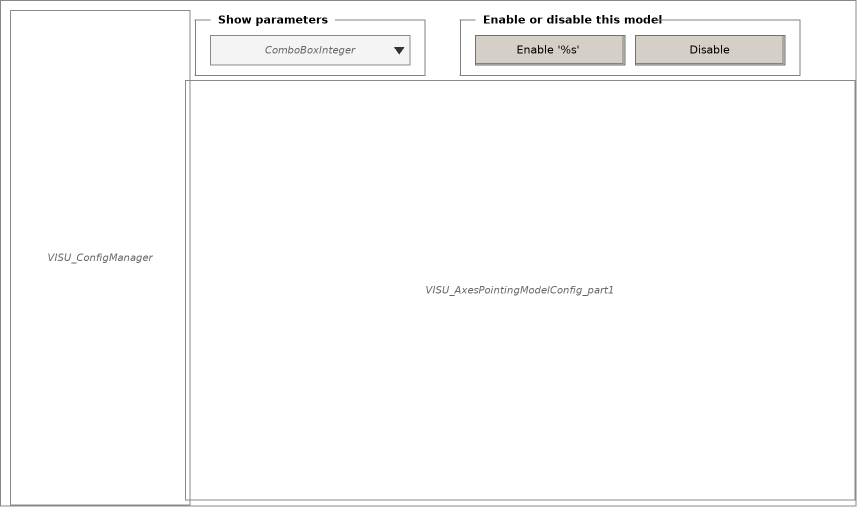
VISUALIZATION VISU_AxesPointingModelSetup  // 857x507
VAR_IN_OUT
    ref : AxesPointingModelSetup;
    widget : AxesPointingModelSetupWidget;
END_VAR
    Polyline (210,20) (195,20) (195,75) (425,75) (425,20) (335,20)
    Frame (10,10 180x495)
        shows VISU_ConfigManager(mgr := ref.parts.configManager, widget := widget.configManager)
    Frame (185,80 670x420), frame switch variable: widget.part
        shows VISU_AxesPointingModelConfig_part1(active := ref.config, editable := ref.editableConfig)
        shows VISU_AxesPointingModelConfig_part2(active := ref.config, editable := ref.editableConfig)
        shows VISU_MeasurementConfig(active := active.temperatures.m2Electronics, editable := editable.temperatures.m2Electronics)
        shows VISU_MeasurementConfig(active := active.temperatures.topTube, editable := editable.temperatures.topTube)
        shows VISU_MeasurementConfig(active := active.temperatures.centreTube, editable := editable.temperatures.centreTube)
        shows VISU_MeasurementConfig(active := active.temperatures.fork, editable := editable.temperatures.fork)
        shows VISU_MeasurementConfig(active := active.temperatures.nasmythAir, editable := editable.temperatures.nasmythAir)
        shows VISU_MeasurementConfig(active := active.temperatures.rem, editable := editable.temperatures.rem)
        shows VISU_MeasurementConfig(active := active.temperatures.rpm, editable := editable.temperatures.rpm)
        shows VISU_MeasurementConfig(active := active.temperatures.hermesTelescopeAdapter, editable := editable.temperatures.hermesTelescopeAdapter)
        shows VISU_MeasurementConfig(active := active.temperatures.topAir, editable := editable.temperatures.topAir)
        shows VISU_MeasurementConfig(active := active.temperatures.insideTube, editable := editable.temperatures.insideTube)
        shows VISU_MeasurementConfig(active := active.relativeHumidities.topAir, editable := editable.relativeHumidities.topAir)
        shows VISU_MeasurementConfig(active := active.relativeHumidities.insideTube, editable := editable.relativeHumidities.insideTube)
        shows VISU_MeasurementConfig(active := active.dewpoints.topAir, editable := editable.dewpoints.topAir)
        shows VISU_MeasurementConfig(active := active.dewpoints.insideTube, editable := editable.dewpoints.insideTube)
        shows VISU_MeasurementConfig(active := active.accelerometers.tube.x, editable := editable.accelerometers.tube.x)
        shows VISU_MeasurementConfig(active := active.accelerometers.tube.y, editable := editable.accelerometers.tube.y)
        shows VISU_AxesConfig_LocalConditions(active := active.localConditions, editable := editable.localConditions)
    ComboBoxInteger (210,35 200x30), variable: widget.part, text list: 'AxesPointingModelSetupPartsTextList'
    Label (480,10 180x20), "Enable or disable this model"
    Polyline (475,20) (460,20) (460,75) (800,75) (800,20) (655,20)
    Button (475,35 150x30), "Enable '%s'", text variable: ref.config.name, input disabled if: widget.enableButtonDisabled
        OnMouseClick: execute { widget.enableButtonPressed := TRUE; }
    Button (635,35 150x30), "Disable", input disabled if: widget.disableButtonDisabled
        OnMouseClick: execute { widget.disableButtonPressed := TRUE; }
    Label (215,10 125x20), "Show parameters"
END_VISUALIZATION

(* stored: Version 1.1.0.1, ProductVersion 3.1.4019.2
   Visu VISU_AxesPointingModelSetup: Id {13323f1a-cf53-488f-8bad-5c9271448a94} *)
